ORGANIZATION_BLOCK Prog1:einfacher_Schalter
BEGIN
NETWORK 1
	LD E0.0
	S A0.0,1
NETWORK 2
  LD E0.1
  R A0.0,1
END_ORGANIZATION_BLOCK
